FUNCTION TryConvert_LWORD_TO_BOOL : BOOL
VAR_INPUT
	in : LWORD;
	out : REFERENCE TO BOOL;
END_VAR

out := LWORD_TO_BOOL(in);
TryConvert_LWORD_TO_BOOL := TRUE;

END_FUNCTION

(* stored: Version 1.1.0.1, ProductVersion 3.1.4024.12
   POU TryConvert_LWORD_TO_BOOL: Id {3f4c0f75-c0a0-415d-bfb7-2acd13d68ad5}, SpecialFunc None *)
